# EPICS autosave request: ADApp/Db/NDPluginTransform_settings.req
$(P)$(R)Name
$(P)$(R)Type1
$(P)$(R)Type2
$(P)$(R)Type3
$(P)$(R)Type4
$(P)$(R)OriginLocation
